TYPE ST_UC_Status_Dummy EXTENDS ST_UC_Status :
STRUCT
	R1_10_UC_Rx_cobID : UDINT;
	R1_10_UC_Rx_data : ARRAY [0..7] OF BYTE;
END_STRUCT
END_TYPE

(* stored: Version 1.1.0.1, ProductVersion 3.1.4024.11
   DUT ST_UC_Status_Dummy: Id {d21820f6-7613-400a-bf05-0f21c13c1357} *)
